(*
Nazwa:			GVL_Recipe
Opis:			Zmienne recepturowe tylko do wizualizacji
Wersja:			v0.2
Data:			2024-02-20
Autor:			AS
Urzadzenia:		
Konfiguracja:	
Info:
Zmiany:
- 20240220 [DP] Poprawki przed nowa wizką
*)

{attribute 'qualified_only'}
VAR_GLOBAL
	(*Legenda dla wizki :
		[H] - Hidden, prawdopodobnie nie potrzebne
		[I] - Info, informacja,
		[L] - Later, do zrobienia później, być może do przerobienia
		Uprawienia:
		brak opisu - operator
		[m] - Meechanik i powyżej
		[t] - Technolog i powyżej
		[s] - Serwis i powyżek
		[a] - Admin			
	*)	

(******BottleSupplySorter********)	
(*******************************BottleSupplySorter Product Type**************************************************************************)	
	//Sorter butelek, typ produktu
	iBottleSorterProductTypeShow												: INT;					// 		Typ produktu
	uiBottleSorterIndexShow														: DINT;					// 		Index butelki 	
	                                                                   
(*******************************BottleSupplySorterHopperTransporter**************************************************************************)	
	//Sorter butelek, transporter zasobnika
	bBottleSorterHopperTransporterEnableShow									: BOOL;					//  	Aktywacja
	iBottleSorterHopperConveyorRunningSpeedSVShow								: INT	:= 5;			// 		Prędkość | [%] (1-100)
	iBottleSorterHopperConveyorEmptyingSpeedSVShow								: INT	:= 7;			// 		Prędkość, opróżnianie	| [%] (1-100)
	iBottleSorterDistanceToFindElementOnTransferConveyorLimitRunningSVShow		: INT	:= 610; 		// 		Odległość do butelek | [mm] (10-10_000)                                  		
	iBottleSorterDistanceToFindElementOnTransferConveyorLimitEmptyingSVShow		: INT	:= 500; 		// 		Odległość do butelek - opróżnianie | [mm] (10-10_000)                                       		

(*******************************BottleSupplySorterTransferTransporter**************************************************************************)
	//Sorter butelek, transporter transferowy	
	bBottleSorterTransferTransporterEnableShow									: BOOL;					// 		Aktywacja
	iBottleSorterTransferConveyorRunningSpeedSVShow								: INT	:= 5;			// 		Prędkość | [%] (1-100)	
	iBottleSorterTransferConveyorEmptyingSpeedSVShow							: INT	:= 7;			// 		Prędkość, opróżnianie | [%] (1-100)
	iBottleSorterDistanceToFindElementOnSupplyConveyorDownstairsLimitSVShow		: INT	:= 600;			// 		Odległość do butelek - stop zasypu | [mm] (10-10_000)
                                                                               
(*******************************BottleSupplySorterSupplyTransporter**************************************************************************)	
	//Sorter butelek, transporter zasypowy
	bBottleSorterSupplyTransporterEnableShow									: BOOL;					// [H] 	Aktywacja
	uiBottleSorterSupplyTransporterRunningSpeedSVShow							: UINT	:= 1_000;		// 		Prędkość | [obr/min] (10-10_000)	
	uiBottleSorterSupplyTransporterEmptingSpeedSVShow							: UINT	:= 1_000;		// 		Prędkość, opróżnianie | [obr/min] (10-10_000)                                                                   
	lrBottleSorterModuloMoveOffsetSVShow										: LREAL;				// 		Kat sprawdzania | [°] (1-360)	                                                                            
	//Logika zasypu - warunek pierwszy	                                                            
	iBottleSorterSensorsCountFirstConditionSVShow								: INT;					// 		Limit butelek
	iBottleSorterSupplyTimeFirstConditionSVShow									: INT;					// 		Czas zasypu | [ms] (10-10_000)                                                                                                    		
	//Logika zasypu - warunek drugi	 	                                                                                       		
	iBottleSorterSensorsCountSecondConditionMinSVShow							: INT;					// 		Limit butelek, min
	iBottleSorterSensorsCountSecondConditionMaxSVShow							: INT;					// 		Limit butelek, max
	iBottleSorterSupplyTimeSecondConditionSVShow								: INT;					// 		Czas zasypu | [ms] (10-10_000)                                                                                                  		
	//Logika zasypu - warunek trzeci 	                                                                                       		
	iBottleSorterSensorsCountThirdConditionSVShow								: INT;					// 		Limit butelek
	iBottleSorterSupplyTimeThirdConditionSVShow									: INT;					// 		Czas zasypu | [ms] (10-10_000)
	                                                                            	
(*******************************BottleSupplySorterWheel**************************************************************************)	
	//Sorter butelek, Stól
	bBottleSorterWeelEnableShow													: BOOL;					// [H]	Aktywacja
	lrBottleSorterWheelSpeedSVShow												: LREAL := 20;			// 		Prędkość | [obr/min] (5-100)	            
	lrBottleSorterWheelEmptyingSpeedSVShow										: LREAL := 30;			// 		Prędkość, opróżnianie | [obr/min] (5-100)	
		
(*******************************BottleSupplySorterBrush**************************************************************************)		
	//Sorter butelek, szczotka
	bBottleSorterBrushEnableShow												: BOOL;					//		Aktywacja
	lrBottleSorterBrushHeightPositionSVShow										: LREAL := 71;			// 		Wysokosc | [mm] (10-200)	
	iBottleSorterBrushRunningSpeedSVShow										: INT; 		 			// 		Prędkość | [%] (1-100)	            
	iBottleSorterBrushEmptyingSpeedSVShow										: INT; 		 			// 		Prędkość, opróżnianie | [%] (1-100)                                                              		         	
	
(*********************************BottleSupplyRobot*******************************************************************)

	//Sorter butelek, robot
	bBottleSorterRobotEnableShow												: BOOL;					// 		Aktywacja     
	nBottleSorterRobotRecipeId													: UDINT;				//		Nr receptury                                                                   
	//Czasy przyssania i oddmuchu                                                                                                                              
	lrBottleSorterRemainingTimeToSuctionShow             						: LREAL;				// 		Wyprzedzenie przyssania | [ms] (0-200)
	lrBottleSorterSuckerSuctionTimeShow											: LREAL;				// 		Czas przyssania	| [ms] (10-1000)
    lrBottleSorterRemainingTimeToRejectShow             						: LREAL;				// 		Wuprzedzenie oddmuchu | [ms] (0-200)
	lrBottleSorterEjectorPulseShow                                       		: LREAL;				// 		Czas oddmuchu	| [ms] (10-1000)			                                                                                                    		                                                                                                        		
	//Pkt. poboru i dokładania                                                                                 		                                                                                                          		
	lrBottleSorterZPickAboveTheBottleSVShow										: LREAL;				// 		Wysokość pobierania butelki
	lrBottleSorterZPickMoveSVShow												: LREAL;				// 		Odległość zjazdu w dół łapanie butelki 	                                                                                               	   		                                                                                     		
	lrBottleSorterSafetyHeightSVShow											: LREAL	:= 150;  		// 		Wysokość obracania chwytaka | [mm] (0-1000)

(*********************************BottleReciever*******************************************************************)

	//Sorter butelek, robot
	bBottleSorterRecieverEnableShow												: BOOL;					// 		Aktywacja   
	bBottleSorterRecieverSlot1EnableShow										: BOOL;					// 		Aktywacja  
	bBottleSorterRecieverSlot2EnableShow										: BOOL;					// 		Aktywacja  
	bBottleSorterRecieverSlot3EnableShow										: BOOL;					// 		Aktywacja  
	lrBottleSorterRecieverHeightPositionSVShow									: LREAL;				// 		Wysokosc | [mm] (10-200)
                                                                   
	lrBottleSorterRecieverSlotPositionSVShow									: LREAL;				
	lrBottleSorterRecieverMiddlePositionSVShow									: LREAL;				
	lrBottleSorterRecieverPuckPositionSVShow									: LREAL;				

END_VAR

(* stored: Version 1.1.0.1, FileIdentifier 164db32f566a473704d1bc097a55c55c3302a66e, FileSignature 1077831301c9a82dd8dd3335cdac44ae6e7986baca8dc26c42a37cca79f40da5944b0a2a9328a45dcb86dec7cd309e38b68d393c834c4b914975bfdbbfc256dab59df4ea117555d12335d01fd9ec74da5f378048e75823070ee15f57d060edc6561eaf8d97fa74876af1d3aecc0cc91426da9f55197518ffe28c3938b037dfb78069d9afd72d09c0a3f9efdd35fb13a0aa193b9831878c143f3ea7aaccb8bf662a91d137d528e7453d7d7f36768ada748e5c599eec2e20736061d3442adf1785aeccb291e0a52460ce5a374a45bf9f761b8ab4e6e6d104c22c0c28df4068159e6d784dc35b3a575451ece94bcfc9cb9b15156bdd0460f9775074ee9cd0a43756
   GVL GVL_Recipe: Id {f7069ba5-8f3f-45eb-97f8-f62e0bd4b8ad} *)
